// TwinCAT 3 PLC project Carrier
// ProgramVersion: 3.1.4024.0
// libraries:
//   Tc2_Standard, * (Beckhoff Automation GmbH)
//   Tc2_System, * (Beckhoff Automation GmbH)
//   Tc3_Module, * (Beckhoff Automation GmbH)
//   VisuSymbols,3.5.10.0,System
// project tree:
//   DUTs/ Buffer_Slots.TcDUT, E_PickerTransitionState.TcDUT, E_PickerFixedState.TcDUT
//   FBs/ FB_Buffer.TcPOU, FB_Picker.TcPOU, FB_Picker_1.TcPOU, FB_Picker_2.TcPOU
//   / GlobalTextList.TcGTLO, PlcTask.TcTTO, Visualization Manager.TcVMO (not stored)
//   GVLs/ GVL.TcGVL
//   POUs/ MAIN.TcPOU
//   VISUs/ Visualization.TcVIS
// real-time tasks:
//   TASK PlcTask: cycle T#10ms, priority 20, ADS port 350

CONFIGURATION Carrier
    RESOURCE PLC ON TwinCAT3
        TASK PlcTask(INTERVAL := T#10ms, PRIORITY := 20);
        PROGRAM MAIN WITH PlcTask : MAIN;
    END_RESOURCE
END_CONFIGURATION

// ---- DUTs/Buffer_Slots.TcDUT
TYPE Buffer_Slots :
STRUCT
	Slot_Full      : BOOL;   //If TRUE there is part in the Buffer Slot
	Serial_Number   : UDINT; //Serial Number of Part in the Buffer Slot
END_STRUCT
END_TYPE

// ---- DUTs/E_PickerTransitionState.TcDUT
{attribute 'qualified_only'}
{attribute 'strict'}
TYPE E_PickerTransitionState :
(

	MoveToPick  := 11,
	Picking     := 12,
	MoveToPlace := 13,
	Placing     := 14
);
END_TYPE

// ---- DUTs/E_PickerFixedState.TcDUT
{attribute 'qualified_only'}
{attribute 'strict'}
TYPE E_PickerFixedState :
(
	Idle        := 0,
	InPickedPos := 1,
	PartPicked 	:= 2,
	InPlacedPos := 3,
	PartPlaced  := 4
);
END_TYPE

// ---- GVLs/GVL.TcGVL
{attribute 'qualified_only'}
VAR_GLOBAL CONSTANT
	Buffer_Size : UINT := 12;
END_VAR

// ---- POUs/MAIN.TcPOU
PROGRAM MAIN
VAR
	
    Buffer_1                   : FB_Buffer;
    Buffer_2                   : FB_Buffer;
	
	Picker_1                   : FB_Picker_1;
	Picker_2                   : FB_Picker_2;
	
	ClearBuffer_1              : BOOL; // Clear Parts Buffer Slots from Buffer_1
	ClearBuffer_2              : BOOL; // Clear Parts Buffer Slots from Buffer_2
	
	Disable_Picker_2 		   : BOOL; //If TRUE Picker_2 finishes current job and remains IDLE at Carrier_Pos (place part from Buffer)
	Disable_Picker_1 		   : BOOL; //IF TRUE Picker_1 finished current job and remains IDLE at Cassette_Pos (pick new part)
	
	//Serial Part Number
	Serial_Number_Generator    : UDINT; //Pseudo New Part Generator; creates Serial for every new part in the cassette
	
	New_Part_Serial_Number     : UDINT; //New Part Serial Number in Cassette (picked from Cassette by Picker_1)
	Carrier_Part_Serial_Number : UDINT; //Latest Carrier Part Serial Number (handed over to Carrier by Picker_2)
	
	
	Clear_Serial_Number        : BOOL; //when TRUE reset Serial_Number_Generator to 0
	
	New_Part_Ack               : BOOL; //When TRUE Picker_1 acknowledges placing of new Part Serial Number on BufferSlot; Picker_2 resets it when picks part
END_VAR


Buffer_1();
Buffer_2();

Picker_1();
Picker_2();


_M_Sequence_Picker1(); // Run Picker_1 Pick from Cassette & Place to Buffer_1/Buffer_2 Sequence
_M_Sequence_Picker2(); // Run Picker_2 Pick from Availble Buffer_1/Buffer_2 Slot & Place to Carrier





IF ClearBuffer_1 THEN        //if TRUE it empties all Buffer_1 Part Slots
	Buffer_1.M_ClearBuffer();
	ClearBuffer_1 := FALSE;
END_IF


IF ClearBuffer_2 THEN      // if TRUE it empties all Buffer_2 Part Slots
	Buffer_2.M_ClearBuffer();
	ClearBuffer_2 := FALSE;
END_IF

IF Disable_Picker_2 THEN  //If TRUE Picker_2 finishes current job and remains IDLE at Carrier
	Picker_2.M_DisablePicker();
ELSE
	Picker_2.M_EnablePicker();
END_IF

IF Disable_Picker_1 THEN //If TRUE Picker_1 finishes current job and remains IDLE at Cassette
	Picker_1.M_DisablePicker();
ELSE
	Picker_1.M_EnablePicker();
END_IF

IF Clear_Serial_Number THEN //If TRUE it resets Serial Part Generator to 0
	Serial_Number_Generator := 0;
	Clear_Serial_Number := FALSE;
END_IF

New_Part_Serial_Number := Serial_Number_Generator; //Sim serial number for every new part

METHOD PRIVATE _M_Sequence_Picker1 : BOOL
VAR_INPUT
END_VAR
IF Picker_1.State = E_PickerFixedState.Idle AND   //If both buffers are empty and both Pickers are idle, Picker1 is picking a part
	Picker_2.State = E_PickerFixedState.Idle AND  //to initiate the pick-place sequence
	Buffer_1.IsEmpty AND Buffer_2.IsEmpty THEN 
	
	Picker_1.M_MoveToPickPos();
END_IF


CASE Picker_1.State OF
	
	E_PickerFixedState.Idle:
	
		IF NOT Picker_1.Disable_Picker THEN 
			Picker_1.M_PickPart();
		END_IF
	
	E_PickerFixedState.InPickedPos:
	
		IF Picker_1.Disable_Picker THEN 
			Picker_1.M_IdleState();
		ELSE
			Picker_1.M_PickPart();
		END_IF
		
		
	E_PickerFixedState.PartPicked:
	
	
		Picker_1.P_TargetPosition_Buffer := 0; //Initialize Buffer Position to zero 
	
		IF (Picker_2.TargetBuffer_Is_2 OR  ((Picker_2.State = E_PickerFixedState.Idle) OR (Picker_2.State >= E_PickerFixedState.InPlacedPos) )) AND NOT Buffer_1.IsFull  THEN 
			
				Picker_1.P_TargetPosition_Buffer := Buffer_1.M_Find_First_Empty_Pos(); //Find  available position in the buffer
				
				IF Picker_1.TargetPosition_Buffer <> 0 THEN 
					Picker_1.M_TargetBuffer_Is_1();   //Picker_1 will go to deliver part to Buffer_1 since either Picker_2 is idle or is busy with Buffer_B
				END_IF
				
		ELSIF ((Picker_2.State = E_PickerFixedState.Idle) OR (Picker_2.State >= E_PickerFixedState.InPlacedPos)) AND NOT Buffer_2.IsFull    THEN 
			
				Picker_1.P_TargetPosition_Buffer := Buffer_2.M_Find_First_Empty_Pos(); //Find position available position in the buffer
		
				IF Picker_1.TargetPosition_Buffer <> 0 THEN 
					Picker_1.M_TargetBuffer_Is_2();   //Picker_1 will go to deliver part to Buffer_1 since either Picker_2 is idle or is busy with Buffer_B
				END_IF
		
		
		
		END_IF
		
		IF NOT New_Part_Ack THEN 
			Serial_Number_Generator := Serial_Number_Generator + 1;
			New_Part_Ack := TRUE;
		END_IF
	
		
		IF  Picker_1.TargetPosition_Buffer <> 0 THEN //If there is valid buffer target position, pass buffer type and the buffer position for the Picker to place the part
			Picker_1.M_MoveToPlacePos(Buffer_1_InUse := Picker_1.TargetBuffer_Is_1, Buffer_Pos := Picker_1.TargetPosition_Buffer   ); //Pseudo code to send the Picker to the respective buffer position (buffer type + buffer position)
		END_IF
		
	
	E_PickerFixedState.InPlacedPos:
		Picker_1.M_PlacePart();
			
	E_PickerFixedState.PartPlaced:
	
		New_Part_Ack := FALSE; //Reset Serial Number Handover Acknowledgement bit
		Picker_1.M_MoveToPickPos();
		
		IF Picker_1.TargetBuffer_Is_1 THEN 
			Buffer_1.M_PlacePartInBuffer(Picker_1.TargetPosition_Buffer,New_Part_Serial_Number);
		ELSE 
			Buffer_2.M_PlacePartInBuffer(Picker_1.TargetPosition_Buffer,New_Part_Serial_Number);
		END_IF
		
	

END_CASE
END_METHOD

METHOD PRIVATE _M_Sequence_Picker2 : BOOL
VAR_INPUT
END_VAR
CASE Picker_2.State OF 
	
	E_PickerFixedState.PartPlaced :
	
		IF Picker_1.TargetBuffer_Is_1 THEN //If Picker_1 is in Buffer_1 then Picker_2 can pick part from Buffer_2 with no Collision Risk
			IF NOT Buffer_2.IsEmpty THEN 
				
				Picker_2.P_TargetPosition_Buffer := Buffer_2.M_Find_First_Occupied_Pos(); //If Buffer_2 has at least one part, find first available location
			
				IF (Picker_2.TargetPosition_Buffer <> 0)  AND (Picker_1.State <= E_PickerFixedState.PartPicked)  THEN //If Buffer returns available valid position ( no zero) then 
					Picker_2.M_TargetBuffer_Is_2();         //set Buffer_2 as target buffer and set to the Picker_2 the position of the buffer 
					Picker_2.M_MoveToPickPos(Buffer_1_InUse:= FALSE , Buffer_Pos := Picker_2.TargetPosition_Buffer );
				
				END_IF
				
			ELSE //If Buffer_1 Is Empty and Picker_1 is Idle then Picker_2 should move to Buffer_2
				Picker_2.P_TargetPosition_Buffer := Buffer_1.M_Find_First_Occupied_Pos(); //If Buffer_2 has at least one part, find first available location
			
				IF (Picker_2.TargetPosition_Buffer <> 0) AND (Picker_1.State <= E_PickerFixedState.PartPicked) THEN //If Buffer returns available valid position ( no zero) then 
					Picker_2.M_TargetBuffer_Is_1();         //set Buffer_2 as target buffer and set to the Picker_2 the position of the buffer 
					Picker_2.M_MoveToPickPos(Buffer_1_InUse:= TRUE , Buffer_Pos := Picker_2.TargetPosition_Buffer );
				
				END_IF
			
			END_IF
			
		ELSIF Picker_1.TargetBuffer_Is_2 AND (Picker_1.State <= E_PickerFixedState.PartPicked)  THEN 
			
			IF NOT Buffer_1.IsEmpty THEN 
				
				Picker_2.P_TargetPosition_Buffer := Buffer_1.M_Find_First_Occupied_Pos(); //If Buffer_2 has at least one part, find first available location
			
				IF Picker_2.TargetPosition_Buffer <> 0 THEN //If Buffer returns available valid position ( no zero) then 
					Picker_2.M_TargetBuffer_Is_1();         //set Buffer_2 as target buffer and set to the Picker_2 the position of the buffer 
					Picker_2.M_MoveToPickPos(Buffer_1_InUse:= TRUE , Buffer_Pos := Picker_2.TargetPosition_Buffer );
				
				END_IF
				
			ELSE //If Buffer_1 Is Empty and Picker_1 is Idle then Picker_2 should move to Buffer_2
				Picker_2.P_TargetPosition_Buffer := Buffer_2.M_Find_First_Occupied_Pos(); //If Buffer_2 has at least one part, find first available location
			
				IF Picker_2.TargetPosition_Buffer <> 0 THEN //If Buffer returns available valid position ( no zero) then 
					Picker_2.M_TargetBuffer_Is_2();         //set Buffer_2 as target buffer and set to the Picker_2 the position of the buffer 
					Picker_2.M_MoveToPickPos(Buffer_1_InUse:= FALSE , Buffer_Pos := Picker_2.TargetPosition_Buffer );
				
				END_IF
			END_IF
			
		
		END_IF
		
		Carrier_Part_Serial_Number := Picker_2.Part_SerialNumber;
		
	E_PickerFixedState.InPickedPos:
		Picker_2.M_PickPart();
	
			
	E_PickerFixedState.PartPicked:
				
	
		Picker_2.P_Part_SerialNumber := SEL(Picker_2.TargetBuffer_Is_1,Buffer_2.M_PickPartFromBuffer(Picker_2.TargetPosition_Buffer),Buffer_1.M_PickPartFromBuffer(Picker_2.TargetPosition_Buffer));
	
		Picker_2.M_MoveToPlacePos();
			
	E_PickerFixedState.InPlacedPos:
	
		IF Picker_2.Disable_Picker THEN 
			Picker_2.M_IdleState();
		ELSE
			Picker_2.M_PlacePart();
		END_IF
			
	E_PickerFixedState.Idle:
	
		IF NOT Picker_2.Disable_Picker THEN 
			Picker_2.M_PlacePart();
		END_IF

END_CASE
END_METHOD

END_PROGRAM

// ---- FBs/FB_Buffer.TcPOU
FUNCTION_BLOCK FB_Buffer

VAR
	BlankBuffer : ARRAY[1..GVL.Buffer_Size] OF BOOL; //Empty Buffer (placeholder array used for comparison)
	FullBuffer  : ARRAY[1..GVL.Buffer_Size] OF BOOL; //Full Buffer (placeholder array used for comparison)
	
	IsEmpty 	: BOOL; //TRUE if Buffer EMPTY (all part slots available)
	IsFull  	: BOOL; //TRUE if Buffer FULL (no available part slots)
	
	Init_Conf   : BOOL := TRUE; //Initialize Bit for Buffer Configuration
	
	TargetPosition_Buffer : INT;  // Position in X axis of Buffer 
END_VAR


VAR PERSISTENT
	Buffer_Slots : ARRAY[1..GVL.Buffer_Size] OF BOOL; (*Buffer Slots state; if ARRAY[Index] = TRUE there is part 
																	  if ARRAY[Index] = FALSE part slot is empty *)
END_VAR

IF Init_Conf THEN 
	MEMSET(ADR(FullBuffer),16#1,SIZEOF(FullBuffer)); //FullBuffer has all slots TRUE; to be used to compare with actual Buffer Places
Init_Conf := FALSE;
END_IF

IsEmpty := MEMCMP(ADR(BlankBuffer),ADR(Buffer_Slots),SIZEOF(BlankBuffer)) = 0; //TRUE if Buffer has zero parts (all slots are empty)

IsFull := MEMCMP(ADR(FullBuffer),ADR(Buffer_Slots),SIZEOF(FullBuffer)) = 0;  //TRUE if Buffer is full (has zero available slots)

METHOD M_ClearBuffer : BOOL
VAR_INPUT
END_VAR

VAR 
	 i : INT;
END_VAR
//Clears all Buffer Slots from parts 
FOR i := 1 TO GVL.Buffer_Size DO 
	Buffer_Slots[i] := FALSE;
END_FOR
END_METHOD

METHOD PUBLIC M_Find_First_Empty_Pos : INT

VAR 
	 i : INT;
END_VAR
//If not zero, it outputs first available empty buffer slot
FOR i := 1 TO GVL.Buffer_Size DO
    IF NOT Buffer_Slots[i] THEN
        M_Find_First_Empty_Pos := i;
        RETURN;
    END_IF
END_FOR
M_Find_First_Empty_Pos := 0;
END_METHOD

METHOD PUBLIC M_Find_First_Occupied_Pos : INT

VAR 
	 i : INT;
END_VAR
//If not zero, it outputs first available occupied buffer slot
FOR i := 1 TO GVL.Buffer_Size DO
    IF  Buffer_Slots[i] THEN
        M_Find_First_Occupied_Pos := i;
        RETURN;
    END_IF
END_FOR
M_Find_First_Occupied_Pos := 0;
END_METHOD

METHOD M_MoveToPos : BOOL
VAR_INPUT
END_VAR
// This call sends the desired X Buffer Coordinate for part pick/place for picker_2/picker_1 respectively
END_METHOD

METHOD PUBLIC M_PickPartFromBuffer : BOOL
VAR_INPUT
	Select_Index : INT;
END_VAR
//Picker_2 is picking part from Buffer Slot at position Select_Index
Buffer_Slots[Select_Index] := FALSE;
END_METHOD

METHOD M_PlacePartInBuffer : BOOL
VAR_INPUT
	Select_Index : INT;
END_VAR
//Picker_1 is placing part in Buffer Slot at position Select_Index
Buffer_Slots[Select_Index] := TRUE;
END_METHOD

PROPERTY P_TargetPosition_Buffer : INT
GET
P_TargetPosition_Buffer := TargetPosition_Buffer;
END_GET
SET
TargetPosition_Buffer := P_TargetPosition_Buffer;
END_SET
END_PROPERTY

END_FUNCTION_BLOCK

// ---- FBs/FB_Picker_1.TcPOU
FUNCTION_BLOCK FB_Picker_1 EXTENDS FB_Picker

SUPER^(); 


_M_Picker_PosY_VISU(); //Compute Y position of Picker_1 to display on VISU

METHOD PRIVATE _M_Picker_PosY_VISU : BOOL
VAR_INPUT
END_VAR
//Used to simulate Picker Y position on VISU based on pixel Y position and Picker State

IF TargetBuffer_Is_1 AND ((State = E_PickerFixedState.InPlacedPos) OR  (State = E_PickerFixedState.PartPlaced)) THEN 
	IF (TargetPosition_Buffer = 1 ) OR (TargetPosition_Buffer = 7 ) THEN 
		Picker_PosY_VISU_Sim := 2238 -530;
	ELSIF (TargetPosition_Buffer = 2 ) OR (TargetPosition_Buffer = 8) THEN	
		Picker_PosY_VISU_Sim := 2238 -477;
	ELSIF (TargetPosition_Buffer = 3 ) OR (TargetPosition_Buffer = 9) THEN	
		Picker_PosY_VISU_Sim := 2238 -411;
	ELSIF (TargetPosition_Buffer = 4 ) OR (TargetPosition_Buffer = 10) THEN	
		Picker_PosY_VISU_Sim := 2238 -329;
	ELSIF (TargetPosition_Buffer = 5 ) OR (TargetPosition_Buffer = 11) THEN	
		Picker_PosY_VISU_Sim := 2238 -265;
	ELSIF (TargetPosition_Buffer = 6 ) OR (TargetPosition_Buffer = 12) THEN	
		Picker_PosY_VISU_Sim := 2238 -199;
	END_IF
	
ELSIF TargetBuffer_Is_2 AND ((State = E_PickerFixedState.InPlacedPos) OR  (State = E_PickerFixedState.PartPlaced)) THEN 
	IF (TargetPosition_Buffer = 1 ) OR (TargetPosition_Buffer = 7 ) THEN 
		Picker_PosY_VISU_Sim := 2238 - 1181;
	ELSIF (TargetPosition_Buffer = 2 ) OR (TargetPosition_Buffer = 8) THEN	
		Picker_PosY_VISU_Sim := 2238 - 1101;
	ELSIF (TargetPosition_Buffer = 3 ) OR (TargetPosition_Buffer = 9) THEN	
		Picker_PosY_VISU_Sim := 2238 - 1033;
	ELSIF (TargetPosition_Buffer = 4 ) OR (TargetPosition_Buffer = 10) THEN	
		Picker_PosY_VISU_Sim := 2238 - 959;
	ELSIF (TargetPosition_Buffer = 5 ) OR (TargetPosition_Buffer = 11) THEN	
		Picker_PosY_VISU_Sim := 2238 - 884;
	ELSIF (TargetPosition_Buffer = 6 ) OR (TargetPosition_Buffer = 12) THEN	
		Picker_PosY_VISU_Sim := 2238 - 822;
	END_IF

ELSIF (State = E_PickerFixedState.InPickedPos) OR  (State = E_PickerFixedState.PartPicked) THEN 
	Picker_PosY_VISU_Sim := 2238;
END_IF

//Picker_PosY_VISU_Sim := 2238;
//TargetPosition_Buffer
END_METHOD

METHOD M_MoveToPickPos : BOOL
VAR_INPUT
END_VAR

Sim_Time(IN := TRUE, PT := T#400mS);

IF Sim_Time.Q THEN       //We assume in 1 seconds we go to Pick position; CassettePos for Mover1, BufferPos for Mover2
	Sim_Time(IN := FALSE);
	State := E_PickerFixedState.InPickedPos;
END_IF
END_METHOD

METHOD M_MoveToPlacePos : BOOL
VAR_INPUT
	Buffer_1_InUse : BOOL; //TRUE If Buffer_1 is Used, FALSE if Buffer_2 is Used by the Picker
	Buffer_Pos : UINT;     // Dictates the Buffer Slot the place handover takes place
END_VAR
//If Picker_1 then PlaceToCarrier; if  Picker_2  PlaceToBuffer
//State := E_MoverTransitionState.Placing;


Sim_Time(IN := TRUE, PT := T#400MS);

IF Sim_Time.Q THEN   //We assume in 1 seconds we go to Pick position; BufferPos for Mover1, CarrierPos for Mover2
	Sim_Time(IN := FALSE);
	State := E_PickerFixedState.InPlacedPos;
END_IF
END_METHOD

END_FUNCTION_BLOCK

// ---- FBs/FB_Picker.TcPOU
FUNCTION_BLOCK FB_Picker
VAR_INPUT
END_VAR
VAR_OUTPUT
END_VAR
VAR
	//Mover State
	State            : INT; (*Current State of Picker (
								Idle        := 0,
								InPickedPos := 1,
								PartPicked 	:= 2,
								InPlacedPos := 3,
								PartPlaced  := 4*)
	
	StatusDisp       : STRING;
	
	//Inputs
	In_VacuumON      : BOOL; //When True means part is detected in vacuum
	
	//Outputs
	Out_Vacuum       : BOOL; //Becomes TRUE to pick part
	Out_Blower       : BOOL; //Becomes TRUE to put part
	
	//Simulation Timer 
	Sim_Time          : TON ;   //Used to simulate feedback for each state to be riched i.e. time it takes to pick/place
	
	TargetBuffer_Is_1 : BOOL;   // Picker is going to use Buffer 1
	TargetBuffer_Is_2 : BOOL;   // Picker is going to use Buffer 2
	TargetPosition_Buffer : INT;  // Position in y axis of Buffer 
	
	Picker_PosY_VISU_Sim : INT; //Position of Picker in Y position simulating Picker in Y position
	
	Disable_Picker : BOOL;
END_VAR


_M_EvaluateDisplayStatus();

METHOD PRIVATE _M_EvaluateDisplayStatus : BOOL
VAR_INPUT
END_VAR
IF State = E_PickerFixedState.PartPicked THEN 
	StatusDisp := 'Part Picked';
ELSIF State = E_PickerFixedState.PartPlaced THEN 
	StatusDisp := 'Part Placed';
ELSIF State = E_PickerFixedState.InPickedPos THEN 
	StatusDisp := 'Picker in Pick Pos';
ELSIF State = E_PickerFixedState.InPlacedPos THEN 
	StatusDisp := 'Picker in Place Pos';
ELSIF State = E_PickerFixedState.Idle THEN 
	StatusDisp := 'Picker is Idle';
END_IF
END_METHOD

METHOD M_DisablePicker : BOOL
VAR_INPUT
END_VAR
Disable_Picker := TRUE;
END_METHOD

METHOD M_EnablePicker : BOOL
VAR_INPUT
END_VAR
Disable_Picker := FALSE;
END_METHOD

METHOD M_PickPart : BOOL
VAR_INPUT
END_VAR
Out_Blower := FALSE;
Out_Vacuum := TRUE;

Sim_Time(IN := Out_Vacuum, PT := T#500MS);


In_VacuumON := Sim_Time.Q; //We assume when Out_vacuum is TRUE, In_Vacuum feedback becomes true after 100ms

//State := E_MoverTransitionState.Picking;



IF In_VacuumON THEN 
	State := E_PickerFixedState.PartPicked;
	Sim_Time(IN := FALSE);
END_IF
END_METHOD

METHOD M_PlacePart : BOOL
VAR_INPUT
END_VAR
Out_Blower := TRUE;
Out_Vacuum := FALSE;

Sim_Time(IN :=  Out_Blower, PT := T#500MS);


In_VacuumON := Sim_Time.Q; //We assume when Out_vacuum is FALSE, In_Vacuum feedback becomes FALSE after 100ms

//State := E_MoverTransitionState.Placing;



IF  In_VacuumON THEN 
	State := E_PickerFixedState.PartPlaced;
	Sim_Time(IN := FALSE);
END_IF
END_METHOD

METHOD M_TargetBuffer_Is_1 : BOOL
VAR_INPUT
END_VAR
TargetBuffer_Is_1 := TRUE;
TargetBuffer_Is_2 := FALSE;
END_METHOD

METHOD M_TargetBuffer_Is_2 : BOOL
VAR_INPUT
END_VAR
TargetBuffer_Is_1 := FALSE;
TargetBuffer_Is_2 := TRUE;
END_METHOD

PROPERTY P_TargetPosition_Buffer : INT
GET
P_TargetPosition_Buffer := TargetPosition_Buffer;
END_GET
SET
TargetPosition_Buffer := P_TargetPosition_Buffer;
END_SET
END_PROPERTY

END_FUNCTION_BLOCK

// ---- FBs/FB_Picker_2.TcPOU
FUNCTION_BLOCK FB_Picker_2 EXTENDS FB_Picker

VAR
	Part_SerialNumber : UDINT;
END_VAR

SUPER^(); 

_M_Picker_PosY_VISU(); //Compute Y position of Picker_1 to display on VISU

METHOD PRIVATE _M_Picker_PosY_VISU : BOOL
VAR_INPUT
END_VAR
IF TargetBuffer_Is_1 AND ((State = E_PickerFixedState.InPickedPos) OR  (State = E_PickerFixedState.PartPicked)) THEN 
	IF (TargetPosition_Buffer = 1 ) OR (TargetPosition_Buffer = 7 ) THEN 
		Picker_PosY_VISU_Sim := 2238 -530;
	ELSIF (TargetPosition_Buffer = 2 ) OR (TargetPosition_Buffer = 8) THEN	
		Picker_PosY_VISU_Sim := 2238 -477;
	ELSIF (TargetPosition_Buffer = 3 ) OR (TargetPosition_Buffer = 9) THEN	
		Picker_PosY_VISU_Sim := 2238 -411;
	ELSIF (TargetPosition_Buffer = 4 ) OR (TargetPosition_Buffer = 10) THEN	
		Picker_PosY_VISU_Sim := 2238 -329;
	ELSIF (TargetPosition_Buffer = 5 ) OR (TargetPosition_Buffer = 11) THEN	
		Picker_PosY_VISU_Sim := 2238 -265;
	ELSIF (TargetPosition_Buffer = 6 ) OR (TargetPosition_Buffer = 12) THEN	
		Picker_PosY_VISU_Sim := 2238 -199;
	END_IF
	
ELSIF TargetBuffer_Is_2 AND ((State = E_PickerFixedState.InPickedPos) OR  (State = E_PickerFixedState.PartPicked)) THEN 
	IF (TargetPosition_Buffer = 1 ) OR (TargetPosition_Buffer = 7 ) THEN 
		Picker_PosY_VISU_Sim := 2238 - 1181;
	ELSIF (TargetPosition_Buffer = 2 ) OR (TargetPosition_Buffer = 8) THEN	
		Picker_PosY_VISU_Sim := 2238 - 1101;
	ELSIF (TargetPosition_Buffer = 3 ) OR (TargetPosition_Buffer = 9) THEN	
		Picker_PosY_VISU_Sim := 2238 - 1033;
	ELSIF (TargetPosition_Buffer = 4 ) OR (TargetPosition_Buffer = 10) THEN	
		Picker_PosY_VISU_Sim := 2238 - 959;
	ELSIF (TargetPosition_Buffer = 5 ) OR (TargetPosition_Buffer = 11) THEN	
		Picker_PosY_VISU_Sim := 2238 - 884;
	ELSIF (TargetPosition_Buffer = 6 ) OR (TargetPosition_Buffer = 12) THEN	
		Picker_PosY_VISU_Sim := 2238 - 822;
	END_IF

ELSIF (State = E_PickerFixedState.InPlacedPos) OR  (State = E_PickerFixedState.PartPlaced) THEN 
	Picker_PosY_VISU_Sim := 810;
END_IF

//Picker_PosY_VISU_Sim := 2238;
//TargetPosition_Buffer
END_METHOD

METHOD M_MoveToPickPos : BOOL
VAR_INPUT
	Buffer_1_InUse : BOOL;
	Buffer_Pos : UINT;
END_VAR

Sim_Time(IN := TRUE, PT := T#1S);

IF Sim_Time.Q THEN       //We assume in 1 seconds we go to Pick position; CassettePos for Mover1, BufferPos for Mover2
	Sim_Time(IN := FALSE);
	State := E_PickerFixedState.InPickedPos;
END_IF
END_METHOD

METHOD M_MoveToPlacePos : BOOL

Sim_Time(IN := TRUE, PT := T#1S);

IF Sim_Time.Q THEN   //We assume in 1 seconds we go to Pick position; BufferPos for Mover1, CarrierPos for Mover2
	Sim_Time(IN := FALSE);
	State := E_PickerFixedState.InPlacedPos;
END_IF
END_METHOD

PROPERTY P_Part_SerialNumber : UDINT
GET
P_Part_SerialNumber := Part_SerialNumber;
END_GET
SET
Part_SerialNumber := P_Part_SerialNumber;
END_SET
END_PROPERTY

END_FUNCTION_BLOCK

// ---- GlobalTextList.TcGTLO
TEXTLIST GlobalTextList
  561 = '%d'
  676 = '%i'
  288 = '%s'
  135 = 'Buffer 1'
  306 = 'Buffer 2'
  566 = 'Carrier'
  856 = 'Cassette'
  202 = 'Clear Buffer 1'
  750 = 'Clear Buffer 2'
  50 = 'Clear Serial Nr'
  93 = 'Disable '
  387 = 'Disable Mover '
  140 = 'Disable Mover 1'
  400 = 'Latest Part Serial Number'
  477 = 'Mover 1'
  160 = 'Mover 2'
  858 = 'Mover State'
  961 = 'Mover1.'
  824 = 'New Part Serial Number'
  574 = 'Picker'
  153 = 'Picker 1'
  802 = 'Picker 2'
  298 = 'Picker State'
  510 = 'State'
END_TEXTLIST

// ---- VISUs/Visualization.TcVIS
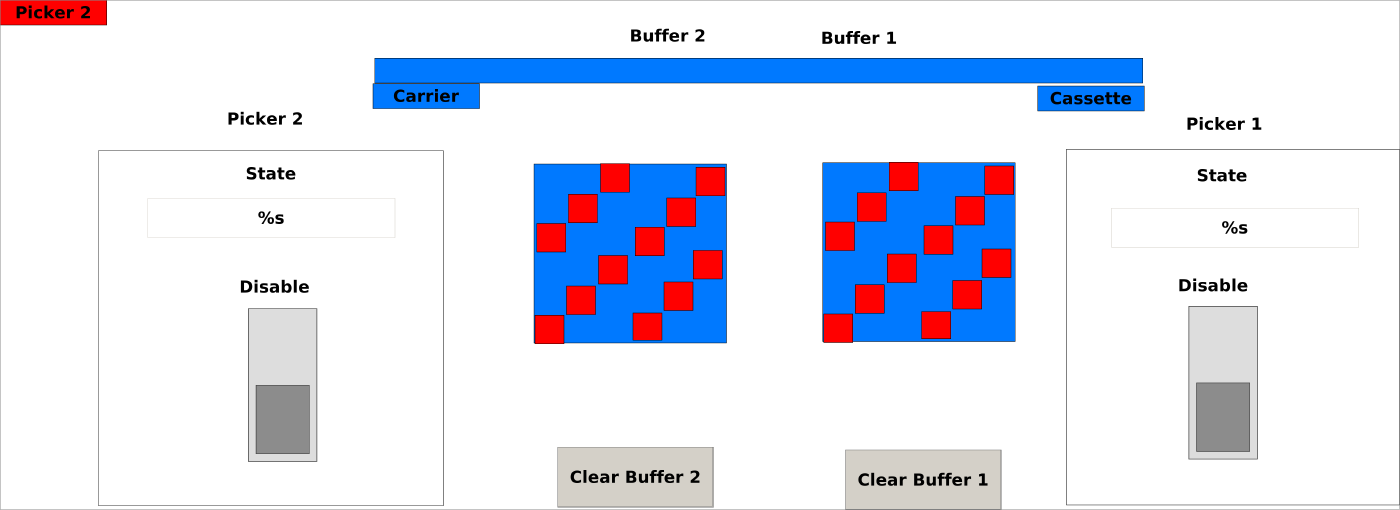
VISUALIZATION Visualization  // 3016x1099
    Rectangle (1150,353 415x386)
    Rectangle (1152,679 63x62), invisible if: NOT MAIN.Buffer_2.Places[1]
    Rectangle (1220,616 63x62), invisible if: NOT MAIN.Buffer_2.Places[2]
    Rectangle (1289,550 63x62), invisible if: NOT MAIN.Buffer_2.Places[3]
    Rectangle (1363,674 63x59), invisible if: NOT MAIN.Buffer_2.Places[4]
    Rectangle (1430,607 63x62), invisible if: NOT MAIN.Buffer_2.Places[5]
    Button (1821,969 336x130), "Clear Buffer 1"
        OnMouseDown: execute { Main.ClearBuffer_1 := TRUE; }
    Button (1201,963 336x130), "Clear Buffer 2"
        OnMouseDown: execute { Main.ClearBuffer_2 := TRUE; }
    Label (1805,278 348x157)
    Label (2283,402 150x115)
    Rectangle (2297,321 719x767)
    Label (2326,462 150x115)
    Textfield (2394,448 533x85), "%s", text variable: MAIN.Picker_1.StatusDisp
    DipSwitch (2470,658 330x333), variable: MAIN.Disable_Picker_1, behaviour: TOGGLE, style: Switch-DipSwitch-Gray
    Label (2433,573 373x84), "Disable"
    Label (2446,336 373x84), "State"
    Rectangle (212,324 743x766)
    Textfield (318,427 533x85), "%s", text variable: MAIN.Picker_2.StatusDisp
    DipSwitch (444,663 330x333), variable: MAIN.Disable_Picker_2, behaviour: TOGGLE, style: Switch-DipSwitch-Gray
    Label (411,576 373x84), "Disable"
    Label (397,332 373x84), "State"
    Label (385,214 373x84), "Picker 2"
    Label (2451,225 373x84), "Picker 1"
    Label (1252,35 373x84), "Buffer 2"
    Label (1664,40 373x84), "Buffer 1"
    Rectangle (1493,539 63x62), invisible if: NOT MAIN.Buffer_2.Places[6]
    Rectangle (1156,481 63x62), invisible if: NOT MAIN.Buffer_2.Places[7]
    Rectangle (1224,418 63x62), invisible if: NOT MAIN.Buffer_2.Places[8]
    Rectangle (1293,352 63x62), invisible if: NOT MAIN.Buffer_2.Places[9]
    Rectangle (1368,489 63x62), invisible if: NOT MAIN.Buffer_2.Places[10]
    Rectangle (1436,426 63x62), invisible if: NOT MAIN.Buffer_2.Places[11]
    Rectangle (1499,360 63x62), invisible if: NOT MAIN.Buffer_2.Places[12]
    Rectangle (1772,350 415x386)
    Rectangle (1774,676 63x62), invisible if: NOT MAIN.Buffer_1.Places[1]
    Rectangle (1842,613 63x62), invisible if: NOT MAIN.Buffer_1.Places[2]
    Rectangle (1911,547 63x62), invisible if: NOT MAIN.Buffer_1.Places[3]
    Rectangle (1985,671 63x59), invisible if: NOT MAIN.Buffer_1.Places[4]
    Rectangle (2052,604 63x62), invisible if: NOT MAIN.Buffer_1.Places[5]
    Rectangle (2115,536 63x62), invisible if: NOT MAIN.Buffer_1.Places[6]
    Rectangle (1778,478 63x62), invisible if: NOT MAIN.Buffer_1.Places[7]
    Rectangle (1846,415 63x62), invisible if: NOT MAIN.Buffer_1.Places[8]
    Rectangle (1915,349 63x62), invisible if: NOT MAIN.Buffer_1.Places[9]
    Rectangle (1990,486 63x62), invisible if: NOT MAIN.Buffer_1.Places[10]
    Rectangle (2058,423 63x62), invisible if: NOT MAIN.Buffer_1.Places[11]
    Rectangle (2121,357 63x62), invisible if: NOT MAIN.Buffer_1.Places[12]
    Rectangle (807,125 1655x54)
    Rectangle (2235,185 230x54), "Cassette"
    Rectangle (803,180 230x54), "Carrier"
    Rectangle (0,0 230x54), "Picker 1"
        p3560616238: MAIN.Picker_1.Picker_PosY_VISU_Sim
    Rectangle (0,0 230x54), "Picker 2"
        p3560616238: MAIN.Picker_2.Picker_PosY_VISU_Sim
END_VISUALIZATION
